{attribute 'qualified_only'}
VAR_GLOBAL
	pS : LREAL := 180;
	pT : LREAL := 1;
	BulkModulus : LREAL := 10000;
	Kv : LREAL := 30 / SQRT(7); 
	DBore : LREAL := 60;
	DRod : LREAL := 40;
	xMax : LREAL := 1.5;
	pi : LREAL := 3.14159265359;
    VA0 : LREAL := 0.2;
	VB0 : LREAL := 0.2;

END_VAR

(* stored: Version 1.1.0.1, ProductVersion 3.1.4024.9
   GVL Param: Id {8cc71902-54f3-4068-b684-2ff92871ee93} *)
